KUKA KRL data list: select.dat

&ACCESS RV
&PARAM TPVW_VERSION = 3.3.5
DEFDAT  SELECT
INT T_NR=0
ENDDAT
